PROGRAM MAIN
VAR
	state : MoveState_t;
	axis1 : AXIS_REF;
	axis2 : AXIS_REF;
	
	moveAbs: MC_MoveAbsolute;
	moveAbsOut: ST_McOutputs;

	power: MC_Power;
	powerOut : ST_McOutputs;
	
	reset: MC_Reset;
	resetOut : ST_McOutputs;
	
	cmd_pos : LREAL;
	cmd_vel : LREAL;
	cmd_acc : LREAL;
	cmd_vel_end : LREAL;
	cmd_need_exe : BOOL;
	
	readActPos: MC_ReadActualPosition;
	readActVel: MC_ReadActualVelocity;
	
	actPosOut : ST_McOutputs;
	actVelOut : ST_McOutputs;
	
	actual_pos : LREAL;
	actual_vel : LREAL;

END_VAR

	
	axis1.ReadStatus();
	
	CASE state OF
		
		MOVESTATE_INIT :
			moveAbs.Execute := FALSE;
			reset.Execute := FALSE;
			power.Enable := FALSE;
			
		MOVESTATE_ENABLE:
			power.Enable := TRUE;
			IF power.Status THEN
				state := MOVESTATE_HOMING;
			ELSIF power.Error THEN
				state := MOVESTATE_ERROR;
			END_IF
		
		MOVESTATE_HOMING:
			state := MOVESTATE_MOVING;
		
		MOVESTATE_MOVING:		
			IF cmd_need_exe THEN
				moveAbs.Position := cmd_pos;
				moveAbs.Velocity := cmd_vel;
				moveAbs.BufferMode := MC_Buffered;
				moveAbs.Execute := TRUE;
				cmd_need_exe := FALSE;			
			END_IF;		
		
			IF moveAbs.Done THEN
				moveAbs.Execute := FALSE;
			ELSIF moveAbs.CommandAborted OR moveAbs.Error THEN
				state := MOVESTATE_ERROR;
			END_IF
			
		MOVESTATE_ERROR :
			IF axis1.Status.Error THEN
				state := MOVESTATE_RESET;
			ELSE
				state := MOVESTATE_INIT;
			END_IF

		MOVESTATE_RESET :
			reset.Execute := TRUE;
			IF reset.Done THEN
				state := MOVESTATE_INIT;
			ELSIF reset.Error THEN
				state := MOVESTATE_INIT;
			END_IF
	END_CASE
	
	
	ActPower();
	ActMove();
	ActReset();
	ActRead();

ACTION ActMove:
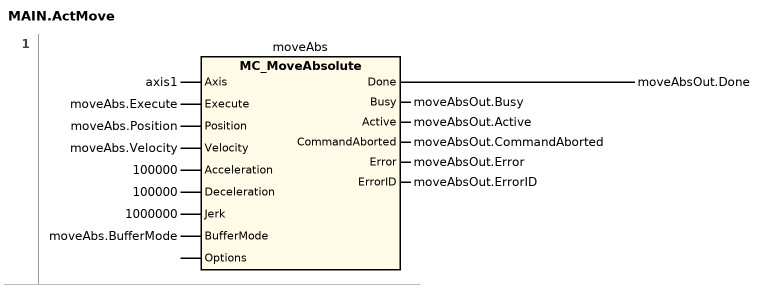
// NETWORK 1
moveAbs(
    Axis := axis1,
    Execute := moveAbs.Execute,
    Position := moveAbs.Position,
    Velocity := moveAbs.Velocity,
    Acceleration := 100000,
    Deceleration := 100000,
    Jerk := 1000000,
    BufferMode := moveAbs.BufferMode,
    Busy => moveAbsOut.Busy,
    Active => moveAbsOut.Active,
    CommandAborted => moveAbsOut.CommandAborted,
    Error => moveAbsOut.Error,
    ErrorID => moveAbsOut.ErrorID); // MC_MoveAbsolute
moveAbsOut.Done := moveAbs.Done;
END_ACTION

ACTION ActPower:
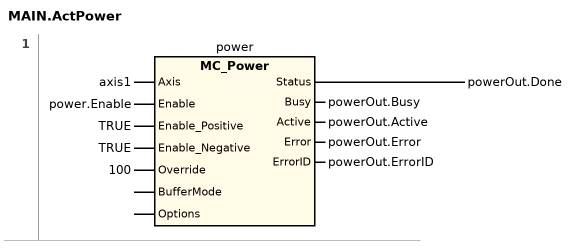
// NETWORK 1
power(
    Axis := axis1,
    Enable := power.Enable,
    Enable_Positive := TRUE,
    Enable_Negative := TRUE,
    Override := 100,
    Busy => powerOut.Busy,
    Active => powerOut.Active,
    Error => powerOut.Error,
    ErrorID => powerOut.ErrorID); // MC_Power
powerOut.Done := power.Status;
END_ACTION

ACTION ActRead:
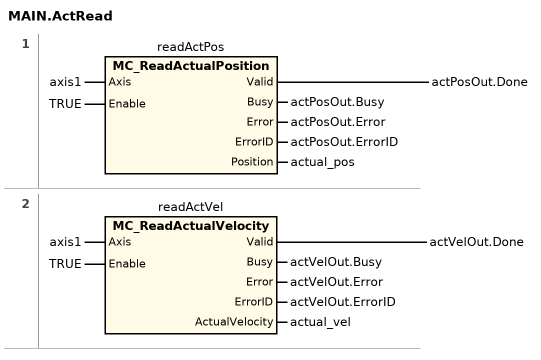
// NETWORK 1
readActPos(
    Axis := axis1,
    Enable := TRUE,
    Busy => actPosOut.Busy,
    Error => actPosOut.Error,
    ErrorID => actPosOut.ErrorID,
    Position => actual_pos); // MC_ReadActualPosition
actPosOut.Done := readActPos.Valid;

// NETWORK 2
readActVel(
    Axis := axis1,
    Enable := TRUE,
    Busy => actVelOut.Busy,
    Error => actVelOut.Error,
    ErrorID => actVelOut.ErrorID,
    ActualVelocity => actual_vel); // MC_ReadActualVelocity
actVelOut.Done := readActVel.Valid;
END_ACTION

ACTION ActReset:
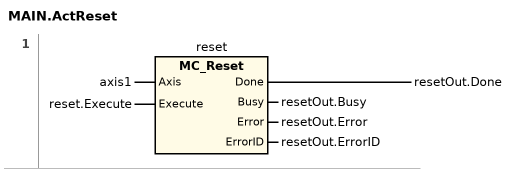
// NETWORK 1
reset(
    Axis := axis1,
    Execute := reset.Execute,
    Busy => resetOut.Busy,
    Error => resetOut.Error,
    ErrorID => resetOut.ErrorID); // MC_Reset
resetOut.Done := reset.Done;
END_ACTION

END_PROGRAM

(* stored: Version 1.1.0.1, ProductVersion 3.1.4020.12
   POU MAIN: Id {0196f569-7f4c-4cc8-b953-20d0a877f80a}, SpecialFunc None
   Action ActMove: Id {247383c3-3462-4c47-9232-c32450d351cb}
   Action ActPower: Id {22a22ddc-1a7b-4ee3-afcd-5be87eff8605}
   Action ActRead: Id {142750ff-8f7d-42cb-81db-ad518e9855c2}
   Action ActReset: Id {64847ba5-ab45-49df-a045-5787b238cbe1} *)
